TYPE (* IEC 61131-3-2.3.3.2 *)
  (* Standard: 61311-3 *)
  (* Version 0.1, 2000-05-16, JHC, Rockwell Automation, File type changed to ".dtp" *)
  (* Version 0.0, 2000-04-18, JHC, Rockwell Automation *)
  (* Compiler header: package fb.rt.ita; *)
  (* Compiler Java IBM VisualAge 3.0 *)
  (* ASN.1 tag PRIVATE 13 *)
  FREQ : REAL := 50;
END_TYPE
